Staubli VAL3: remMovAZELRA.pgx

program remMovAZELRA(string& sArgs[] (dimensions=1), string& sReturn[] (dimensions=1))
  local bool bOk
  local num nAzi
  local num nEle
  local num nLoop
  local num nRad
  local num nVal
  local string sArgsLoop
begin
  // Move to a specified point in spherical coordinates
  //
  // Arguments are "AZ EL RA"
  //
  logMsg("call remMovAZELRA")
  //break down our 3 args and make sure they are numbers
  nLoop=0
  sArgsLoop=sArgs
  while nLoop<3
    sArgsLoop=toNum(sArgsLoop,nVal,bOk)
    if bOk
      switch nLoop
        case 0
          nAzi=nVal
        break
        case 1
          nEle=nVal
        break
        case 2
          nRad=nVal
        break
      endSwitch
      nLoop=nLoop+1
    else
      call remErrNum("MOVAZELRA",sArgs,sReturn)
      return
    endIf
  endWhile
  call remMovSph(nAzi,nEle,nRad,sReturn)
end
